Staubli VAL3: key_check.pgx

program key_check(string x_sString_show (dimensions=1))
begin
  userPage(sScreen_ppShelf)
  title(sScreen_ppShelf,x_sString_show)
  gotoxy(sScreen_ppShelf,0,6)
  putln(sScreen_ppShelf,"Press any key")
  //anykey
  get(sScreen_ppShelf)
  cls(sScreen_ppShelf)
end
